{attribute 'qualified_only'}
VAR_GLOBAL

		HHSwitch	:	BOOL;
		HSwitch		:	BOOL;
		
		LLSwicth	:	BOOL;
		LSwitch		:	BOOL;
		
		Pump		:	BOOL;
		Valve		:	BOOL;
		
		YellowLED	:	BOOL;
		RedLED		:	BOOL;
		BlueLED		:	BOOL;
		
END_VAR

(* stored: Version 1.1.0.1, ProductVersion 3.1.4024.9
   GVL Pump: Id {7b84e801-325e-423b-a5ef-e48e6b8e0efb} *)
